TYPE TYP_DC_MOTOR_HW_OUT :
STRUCT
	Direction AT %Q* : BOOL;
	Run AT %Q* : BOOL;
END_STRUCT
END_TYPE

(* stored: Version 1.1.0.1, ProductVersion 3.1.4024.12
   DUT TYP_DC_MOTOR_HW_OUT: Id {bb137287-10b7-42f5-9cfe-6c9f2786dfd3} *)
